// TwinCAT 3 PLC project plc_kfe_xgmd_vac
// ProgramVersion: 3.1.4022.3
// libraries:
//   L2SI Vacuum Library, * (SLAC)
//   LCLS General, * (SLAC)
//   Tc2_ControllerToolbox, * (Beckhoff Automation GmbH)
//   Tc2_MC2, * (Beckhoff Automation GmbH)
//   Tc2_Standard, * (Beckhoff Automation GmbH)
//   Tc2_System, * (Beckhoff Automation GmbH)
//   Tc2_Utilities, * (Beckhoff Automation GmbH)
//   Tc3_Module, * (Beckhoff Automation GmbH)
// project tree:
//   DUTs/ E_GasType.TcDUT, E_HomeState.TcDUT, E_MoveState.TcDUT (not stored), ST_HV.TcDUT (not stored), ST_VGP.TcDUT
//   GVLs/ GVL_Devices.TcGVL (not stored), GVL_GMD.TcGVL (not stored), GVL_VARIABLES.TcGVL (not stored)
//   / PlcTask.TcTTO (not stored)
//   POUs/ FB_HighVoltage.TcPOU, FB_VGP.TcPOU, MAIN.TcPOU (not stored), PRG_DIAGNOSTIC.TcPOU (not stored), PRG_Gas_Selection.TcPOU, PRG_GMD.TcPOU (not stored), PRG_HV_ILK.TcPOU (not stored), PRG_INJ.TcPOU, PRG_PressureControl.TcPOU (not stored), PRG_Purge.TcPOU, PRG_VGP.TcPOU
// real-time tasks:
//   TASK PlcTask: cycle T#10ms, priority 20, ADS port 350
//   TASK SimTask: cycle T#5ms, priority 21, ADS port 351
// motion (NC):
//   TASK NC-Task 1 SAF: cycle T#2ms, priority 4, ADS port 501
//   TASK NC-Task 1 SVB: cycle T#10ms, priority 8, ADS port 511
//   AXIS VGP_50 (id 1)
//     General: UnitName=step
//     Velo: Maximum=21000
//     OtherSettings: AllowMotionCmdToSlave=true
//     encoder EncType=4
//       EncPara: ScaleFactorNumerator=0.0390625, Inverse=true, MaxCount=#x0000ffff
//         SoftEndMinControl: Enable=true, Range=-15
//         SoftEndMaxControl: Enable=true, Range=1670
//         Inc: RefSoftSyncMask=#x0000ffff
//     drive DrvType=24
//       Analog: VeloReferenz=2000, ScaleFactorActTorque=0.1
//       TimeComp: TaskDelayCycles=1
//     controller CtrType=1
//       CtrPara: PriorControlFactor=1
//         PosDiffControl: Range=50
//         Observer: BandWidth=20
// I/O:
//   DEVICE Device 1 (EtherCAT), AmsNetId 5.62.5.76.2.1
//     EK1200_00_00 [EK1200-5000 EtherCAT Power supply (2A E-Bus)]
//       EL2202_00_01 [EL2202 2Ch. Dig. Output 24V, 0.5A]
//       EL3064_00_02 [EL3064 4Ch. Ana. Input 0-10V]
//       EL1008 [EL1008 8Ch. Dig. Input 24V, 3ms]
//       Term 28 (EL2008) [EL2008 8Ch. Dig. Output 24V, 0.5A]
//       Term 29 (EL2794) [EL2794 4Ch. Dig. Output 24V AC/DC, 2A, short-circuit-proof]
//       Term 30 (EL6695) [EL6695 EtherCAT Bridge terminal (Primary)]
//       Term 31 (EL6695) [EL6695 EtherCAT Bridge terminal (Primary)]
//       Term 32 (EK1110) [EK1110 EtherCAT extension]
//     EK1100_01_00 [EK1100 EtherCAT Coupler (2A E-Bus)]
//       EL3068_01_01 [EL3068 8Ch. Ana. Input 0-10V]
//       EL2794_01_02 [EL2794 4Ch. Dig. Output 24V AC/DC, 2A, short-circuit-proof]
//       EL2794_01_04 [EL2794 4Ch. Dig. Output 24V AC/DC, 2A, short-circuit-proof]
//       EL3068_01_05 [EL3068 8Ch. Ana. Input 0-10V]
//       EL3068_01_06 [EL3068 8Ch. Ana. Input 0-10V]
//       EL2794_01_07 [EL2794 4Ch. Dig. Output 24V AC/DC, 2A, short-circuit-proof]
//       EL2794_01_09 [EL2794 4Ch. Dig. Output 24V AC/DC, 2A, short-circuit-proof]
//       EL3068_01_10 [EL3068 8Ch. Ana. Input 0-10V]
//       EL3068_01_11 [EL3068 8Ch. Ana. Input 0-10V]
//       EL2794_01_12 [EL2794 4Ch. Dig. Output 24V AC/DC, 2A, short-circuit-proof]
//       EL2794_01_14 [EL2794 4Ch. Dig. Output 24V AC/DC, 2A, short-circuit-proof]
//       EL3068_01_15 [EL3068 8Ch. Ana. Input 0-10V]
//       EK1110_01_16 [EK1110 EtherCAT extension]
//     EK1100_02_00 [EK1100 EtherCAT Coupler (2A E-Bus)]
//       EL2004_02_01 [EL2004 4Ch. Dig. Output 24V, 0.5A]
//       EL1004_02_02 [EL1004 4Ch. Dig. Input 24V, 3ms]
//       EL2004_02_03 [EL2004 4Ch. Dig. Output 24V, 0.5A]
//       EL1088_02_04 [EL1088 8Ch. Dig. Input 24V, 3ms, negative]
//       EL2004_02_05 [EL2004 4Ch. Dig. Output 24V, 0.5A]
//       EL1088_02_06 [EL1088 8Ch. Dig. Input 24V, 3ms, negative]
//       EL2004_02_07 [EL2004 4Ch. Dig. Output 24V, 0.5A]
//       EL1004_02_08 [EL1004 4Ch. Dig. Input 24V, 3ms]
//       EL2004_02_09 [EL2004 4Ch. Dig. Output 24V, 0.5A]
//       EL1088_02_10 [EL1088 8Ch. Dig. Input 24V, 3ms, negative]
//       EL2004_02_11 [EL2004 4Ch. Dig. Output 24V, 0.5A]
//       EL1004_02_13 [EL1004 4Ch. Dig. Input 24V, 3ms]
//       EL2004_02_14 [EL2004 4Ch. Dig. Output 24V, 0.5A]
//       EL1088_02_15 [EL1088 8Ch. Dig. Input 24V, 3ms, negative]
//       EL2004_02_16 [EL2004 4Ch. Dig. Output 24V, 0.5A]
//       EL1004_02_17 [EL1004 4Ch. Dig. Input 24V, 3ms]
//       EL3064_02_18 [EL3064 4Ch. Ana. Input 0-10V]
//       EL1008_02_20 [EL1008 8Ch. Dig. Input 24V, 3ms]
//       EL2008_02_22 [EL2008 8Ch. Dig. Output 24V, 0.5A]
//       EL2794_02_23 [EL2794 4Ch. Dig. Output 24V AC/DC, 2A, short-circuit-proof]
//       EL1004_02_24 [EL1004 4Ch. Dig. Input 24V, 3ms]
//       EL2794_02_25 [EL2794 4Ch. Dig. Output 24V AC/DC, 2A, short-circuit-proof]
//       Term 70 (EL9011) [EL9011 End Terminal]
//     EK1100_03_00 (EK1100) [EK1100 EtherCAT Coupler (2A E-Bus)]
//       EL4004_03_01 [EL4004 4Ch. Ana. Output 0-10V, 12bit]
//       EL7041_03_02 [EL7041 1Ch. Stepper motor output stage (50V, 5A)]
//       EL5101_03_03 [EL5101 1Ch. Inc. Encoder 5V]
//       EL1004_03_04 [EL1004 4Ch. Dig. Input 24V, 3ms]
//       EL2004_03_05 [EL2004 4Ch. Dig. Output 24V, 0.5A]
//       EL2004_03_06 [EL2004 4Ch. Dig. Output 24V, 0.5A]
//       EL2004_03_07 [EL2004 4Ch. Dig. Output 24V, 0.5A]
//       EL3202_03_08 [EL3202 2Ch. Ana. Input PT100 (RTD)]
//       EL3174_03_09 [EL3174-0002 4Ch. Ana. Input +/-10V, +/-20mA 16 Bit, Isolated Channels]
// variable links:
//   NC-Task 1 SAF/Axes/VGP_50 <-> Device 1 (EtherCAT)/EK1100_03_00 (EK1100)/EL5101_03_03
//     Enc/Inputs/In/nDataIn1[0] <-> ENC Status compact/Counter value
//     Enc/Inputs/In/nDataIn2[0] <-> ENC Status compact/Latch value
//     Enc/Inputs/In/nState1 @bit 4 <-> ENC Status compact/Status/Counter overflow
//     Enc/Inputs/In/nState1 @bit 3 <-> ENC Status compact/Status/Counter underflow
//     Enc/Inputs/In/nState1 @bit 7 <-> ENC Status compact/Status/Extrapolation stall
//     Enc/Inputs/In/nState1 <-> ENC Status compact/Status/Latch C valid
//     Enc/Inputs/In/nState1 @bit 1 <-> ENC Status compact/Status/Latch extern valid
//     Enc/Inputs/In/nState1 @bit 6 <-> ENC Status compact/Status/Open circuit
//     Enc/Inputs/In/nState1 @bit 2 <-> ENC Status compact/Status/Set counter done
//     Enc/Inputs/In/nState1 @bit 5 <-> ENC Status compact/Status/Status of input status
//     Enc/Inputs/In/nState2 @bit 4 <-> ENC Status compact/Status/Status of extern latch
//     Enc/Inputs/In/nState2 <-> ENC Status compact/Status/Status of input A
//     Enc/Inputs/In/nState2 @bit 1 <-> ENC Status compact/Status/Status of input B
//     Enc/Inputs/In/nState2 @bit 2 <-> ENC Status compact/Status/Status of input C
//     Enc/Inputs/In/nState2 @bit 3 <-> ENC Status compact/Status/Status of input gate
//     Enc/Inputs/In/nState2 @bit 5 <-> ENC Status compact/Status/Sync error
//     Enc/Inputs/In/nState2 @bit 6 <-> ENC Status compact/Status/TxPDO State
//     Enc/Inputs/In/nState2 @bit 7 <-> ENC Status compact/Status/TxPDO Toggle
//     Enc/Inputs/In/nState4 @bit 1 <-> WcState/InputToggle
//     Enc/Inputs/In/nState4 <-> WcState/WcState
//     Enc/Outputs/Out/nCtrl1 <-> ENC Control compact/Control/Enable latch C
//     Enc/Outputs/Out/nCtrl1 @bit 3 <-> ENC Control compact/Control/Enable latch extern on negative edge
//     Enc/Outputs/Out/nCtrl1 @bit 1 <-> ENC Control compact/Control/Enable latch extern on positive edge
//     Enc/Outputs/Out/nCtrl1 @bit 2 <-> ENC Control compact/Control/Set counter
//     Enc/Outputs/Out/nDataOut1[0] <-> ENC Control compact/Set counter value
//   NC-Task 1 SAF/Axes/VGP_50 <-> Device 1 (EtherCAT)/EK1100_03_00 (EK1100)/EL7041_03_02
//     Drive/Inputs/In/nState1 @bit 3 <-> STM Status/Status/Error
//     Drive/Inputs/In/nState1 @bit 5 <-> STM Status/Status/Moving negative
//     Drive/Inputs/In/nState1 @bit 4 <-> STM Status/Status/Moving positive
//     Drive/Inputs/In/nState1 @bit 1 <-> STM Status/Status/Ready
//     Drive/Inputs/In/nState1 <-> STM Status/Status/Ready to enable
//     Drive/Inputs/In/nState1 @bit 6 <-> STM Status/Status/Torque reduced
//     Drive/Inputs/In/nState1 @bit 2 <-> STM Status/Status/Warning
//     Drive/Inputs/In/nState2 @bit 3 <-> STM Status/Status/Digital input 1
//     Drive/Inputs/In/nState2 @bit 4 <-> STM Status/Status/Digital input 2
//     Drive/Inputs/In/nState2 @bit 5 <-> STM Status/Status/Sync error
//     Drive/Inputs/In/nState2 @bit 7 <-> STM Status/Status/TxPDO Toggle
//     Drive/Inputs/In/nState4 @bit 1 <-> WcState/InputToggle
//     Drive/Inputs/In/nState4 <-> WcState/WcState
//     Drive/Outputs/Out/nCtrl1 <-> STM Control/Control/Enable
//     Drive/Outputs/Out/nCtrl1 @bit 2 <-> STM Control/Control/Reduce torque
//     Drive/Outputs/Out/nCtrl1 @bit 1 <-> STM Control/Control/Reset
//     Drive/Outputs/Out/nDataOut2[0] <-> STM Velocity/Velocity
//   plc_kfe_xgmd_vac/plc_kfe_xgmd_vac Instance <-> Device 1 (EtherCAT)/EK1100_01_00/EL2794_01_02
//     PlcTask Outputs/GVL_GMD.fb_EM2K0_XGMD_GCC_10.q_xHV_DIS <-> Channel 1/Output
//     PlcTask Outputs/GVL_GMD.fb_EM2K0_XGMD_GCC_20.q_xHV_DIS <-> Channel 2/Output
//     PlcTask Outputs/GVL_GMD.fb_EM2K0_XGMD_GCC_30.q_xHV_DIS <-> Channel 3/Output
//   plc_kfe_xgmd_vac/plc_kfe_xgmd_vac Instance <-> Device 1 (EtherCAT)/EK1100_01_00/EL2794_01_04
//     PlcTask Outputs/GVL_GMD.fb_EM2K0_XGMD_GCC_40.q_xHV_DIS <-> Channel 1/Output
//     PlcTask Outputs/GVL_GMD.fb_EM2K0_XGMD_GCC_50.q_xHV_DIS <-> Channel 2/Output
//   plc_kfe_xgmd_vac/plc_kfe_xgmd_vac Instance <-> Device 1 (EtherCAT)/EK1100_01_00/EL2794_01_07
//     PlcTask Outputs/GVL_GMD.fb_EM2K0_XGMD_GCC_60.q_xHV_DIS <-> Channel 1/Output
//     PlcTask Outputs/GVL_GMD.fb_EM2K0_XGMD_GCC_70.q_xHV_DIS <-> Channel 2/Output
//     PlcTask Outputs/GVL_GMD.fb_EM2K0_XGMD_GCC_80.q_xHV_DIS <-> Channel 3/Output
//   plc_kfe_xgmd_vac/plc_kfe_xgmd_vac Instance <-> Device 1 (EtherCAT)/EK1100_01_00/EL2794_01_09
//     PlcTask Outputs/GVL_GMD.fb_EM2K0_XGMD_GCC_90.q_xHV_DIS <-> Channel 1/Output
//   plc_kfe_xgmd_vac/plc_kfe_xgmd_vac Instance <-> Device 1 (EtherCAT)/EK1100_01_00/EL3068_01_01
//     PlcTask Inputs/GVL_GMD.fb_EM2K0_XGMD_GCC_10.i_iPRESS_R <-> AI Standard Channel 1/Value
//     PlcTask Inputs/GVL_GMD.fb_EM2K0_XGMD_GCC_20.i_iPRESS_R <-> AI Standard Channel 3/Value
//     PlcTask Inputs/GVL_GMD.fb_EM2K0_XGMD_GCC_30.i_iPRESS_R <-> AI Standard Channel 5/Value
//   plc_kfe_xgmd_vac/plc_kfe_xgmd_vac Instance <-> Device 1 (EtherCAT)/EK1100_01_00/EL3068_01_05
//     PlcTask Inputs/GVL_GMD.fb_EM2K0_XGMD_GCC_40.i_iPRESS_R <-> AI Standard Channel 1/Value
//     PlcTask Inputs/GVL_GMD.fb_EM2K0_XGMD_GCC_50.i_iPRESS_R <-> AI Standard Channel 3/Value
//     PlcTask Inputs/GVL_GMD.fb_EM2K0_XGMD_GPI_10.i_iPRESS_R <-> AI Standard Channel 5/Value
//     PlcTask Inputs/GVL_GMD.fb_EM2K0_XGMD_GPI_90.i_iPRESS_R <-> AI Standard Channel 6/Value
//   plc_kfe_xgmd_vac/plc_kfe_xgmd_vac Instance <-> Device 1 (EtherCAT)/EK1100_01_00/EL3068_01_06
//     PlcTask Inputs/GVL_GMD.fb_EM2K0_XGMD_GCC_60.i_iPRESS_R <-> AI Standard Channel 1/Value
//     PlcTask Inputs/GVL_GMD.fb_EM2K0_XGMD_GCC_70.i_iPRESS_R <-> AI Standard Channel 3/Value
//     PlcTask Inputs/GVL_GMD.fb_EM2K0_XGMD_GCC_80.i_iPRESS_R <-> AI Standard Channel 5/Value
//   plc_kfe_xgmd_vac/plc_kfe_xgmd_vac Instance <-> Device 1 (EtherCAT)/EK1100_01_00/EL3068_01_10
//     PlcTask Inputs/GVL_GMD.fb_EM2K0_XGMD_GCC_90.i_iPRESS_R <-> AI Standard Channel 1/Value
//     PlcTask Inputs/GVL_GMD.fb_EM2K0_XGMD_GPI_50.i_iPRESS_R <-> AI Standard Channel 5/Value
//   plc_kfe_xgmd_vac/plc_kfe_xgmd_vac Instance <-> Device 1 (EtherCAT)/EK1100_02_00/EL1004_02_02
//     PlcTask Inputs/GVL_GMD.fb_EM2K0_XGMD_VRC_10.i_xClsLS <-> Channel 2/Input
//     PlcTask Inputs/GVL_GMD.fb_EM2K0_XGMD_VRC_20.i_xClsLS <-> Channel 4/Input
//     PlcTask Inputs/GVL_GMD.fb_EM2K0_XGMD_VRC_10.i_xOpnLS <-> Channel 1/Input
//     PlcTask Inputs/GVL_GMD.fb_EM2K0_XGMD_VRC_20.i_xOpnLS <-> Channel 3/Input
//   plc_kfe_xgmd_vac/plc_kfe_xgmd_vac Instance <-> Device 1 (EtherCAT)/EK1100_02_00/EL1004_02_08
//     PlcTask Inputs/GVL_GMD.fb_EM2K0_XGMD_VRC_30.i_xClsLS <-> Channel 2/Input
//     PlcTask Inputs/GVL_GMD.fb_EM2K0_XGMD_VRC_40.i_xClsLS <-> Channel 4/Input
//     PlcTask Inputs/GVL_GMD.fb_EM2K0_XGMD_VRC_30.i_xOpnLS <-> Channel 1/Input
//     PlcTask Inputs/GVL_GMD.fb_EM2K0_XGMD_VRC_40.i_xOpnLS <-> Channel 3/Input
//   plc_kfe_xgmd_vac/plc_kfe_xgmd_vac Instance <-> Device 1 (EtherCAT)/EK1100_02_00/EL1004_02_13
//     PlcTask Inputs/GVL_GMD.fb_EM2K0_XGMD_VRC_60.i_xClsLS <-> Channel 2/Input
//     PlcTask Inputs/GVL_GMD.fb_EM2K0_XGMD_VRC_70.i_xClsLS <-> Channel 4/Input
//     PlcTask Inputs/GVL_GMD.fb_EM2K0_XGMD_VRC_60.i_xOpnLS <-> Channel 1/Input
//     PlcTask Inputs/GVL_GMD.fb_EM2K0_XGMD_VRC_70.i_xOpnLS <-> Channel 3/Input
//   plc_kfe_xgmd_vac/plc_kfe_xgmd_vac Instance <-> Device 1 (EtherCAT)/EK1100_02_00/EL1004_02_17
//     PlcTask Inputs/GVL_GMD.fb_EM2K0_XGMD_VRC_80.i_xClsLS <-> Channel 2/Input
//     PlcTask Inputs/GVL_GMD.fb_EM2K0_XGMD_VRC_90.i_xClsLS <-> Channel 4/Input
//     PlcTask Inputs/GVL_GMD.fb_EM2K0_XGMD_VRC_80.i_xOpnLS <-> Channel 1/Input
//     PlcTask Inputs/GVL_GMD.fb_EM2K0_XGMD_VRC_90.i_xOpnLS <-> Channel 3/Input
//   plc_kfe_xgmd_vac/plc_kfe_xgmd_vac Instance <-> Device 1 (EtherCAT)/EK1100_02_00/EL1004_02_24
//     PlcTask Inputs/GVL_GMD.fb_EM2K0_XGMD_PRT_50.i_xAlarmOK <-> Channel 2/Input
//     PlcTask Inputs/GVL_GMD.fb_EM2K0_XGMD_PRT_50.i_xIsRun <-> Channel 1/Input
//   plc_kfe_xgmd_vac/plc_kfe_xgmd_vac Instance <-> Device 1 (EtherCAT)/EK1100_02_00/EL1088_02_04
//     PlcTask Inputs/GVL_GMD.fb_EM2K0_XGMD_PTM_10.i_xAtSpd <-> Channel 1/Input
//     PlcTask Inputs/GVL_GMD.fb_EM2K0_XGMD_PTM_20.i_xAtSpd <-> Channel 3/Input
//     PlcTask Inputs/GVL_GMD.fb_EM2K0_XGMD_PTM_10.i_xFault <-> Channel 2/Input
//     PlcTask Inputs/GVL_GMD.fb_EM2K0_XGMD_PTM_20.i_xFault <-> Channel 4/Input
//   plc_kfe_xgmd_vac/plc_kfe_xgmd_vac Instance <-> Device 1 (EtherCAT)/EK1100_02_00/EL1088_02_06
//     PlcTask Inputs/GVL_GMD.fb_EM2K0_XGMD_PTM_30.i_xAtSpd <-> Channel 1/Input
//     PlcTask Inputs/GVL_GMD.fb_EM2K0_XGMD_PTM_40.i_xAtSpd <-> Channel 3/Input
//     PlcTask Inputs/GVL_GMD.fb_EM2K0_XGMD_PTM_50.i_xAtSpd <-> Channel 5/Input
//     PlcTask Inputs/GVL_GMD.fb_EM2K0_XGMD_PTM_30.i_xFault <-> Channel 2/Input
//     PlcTask Inputs/GVL_GMD.fb_EM2K0_XGMD_PTM_40.i_xFault <-> Channel 4/Input
//     PlcTask Inputs/GVL_GMD.fb_EM2K0_XGMD_PTM_50.i_xFault <-> Channel 6/Input
//   plc_kfe_xgmd_vac/plc_kfe_xgmd_vac Instance <-> Device 1 (EtherCAT)/EK1100_02_00/EL1088_02_10
//     PlcTask Inputs/GVL_GMD.fb_EM2K0_XGMD_PTM_60.i_xAtSpd <-> Channel 1/Input
//     PlcTask Inputs/GVL_GMD.fb_EM2K0_XGMD_PTM_70.i_xAtSpd <-> Channel 3/Input
//     PlcTask Inputs/GVL_GMD.fb_EM2K0_XGMD_PTM_60.i_xFault <-> Channel 2/Input
//     PlcTask Inputs/GVL_GMD.fb_EM2K0_XGMD_PTM_70.i_xFault <-> Channel 4/Input
//   plc_kfe_xgmd_vac/plc_kfe_xgmd_vac Instance <-> Device 1 (EtherCAT)/EK1100_02_00/EL1088_02_15
//     PlcTask Inputs/GVL_GMD.fb_EM2K0_XGMD_PTM_80.i_xAtSpd <-> Channel 1/Input
//     PlcTask Inputs/GVL_GMD.fb_EM2K0_XGMD_PTM_90.i_xAtSpd <-> Channel 3/Input
//     PlcTask Inputs/GVL_GMD.fb_EM2K0_XGMD_PTM_80.i_xFault <-> Channel 2/Input
//     PlcTask Inputs/GVL_GMD.fb_EM2K0_XGMD_PTM_90.i_xFault <-> Channel 4/Input
//   plc_kfe_xgmd_vac/plc_kfe_xgmd_vac Instance <-> Device 1 (EtherCAT)/EK1100_02_00/EL2004_02_01
//     PlcTask Outputs/GVL_GMD.fb_EM2K0_XGMD_VRC_10.q_xOPN_DO <-> Channel 1/Output
//     PlcTask Outputs/GVL_GMD.fb_EM2K0_XGMD_VRC_20.q_xOPN_DO <-> Channel 3/Output
//   plc_kfe_xgmd_vac/plc_kfe_xgmd_vac Instance <-> Device 1 (EtherCAT)/EK1100_02_00/EL2004_02_03
//     PlcTask Outputs/GVL_GMD.fb_EM2K0_XGMD_PTM_10.q_RunDO <-> Channel 1/Output
//     PlcTask Outputs/GVL_GMD.fb_EM2K0_XGMD_PTM_20.q_RunDO <-> Channel 2/Output
//   plc_kfe_xgmd_vac/plc_kfe_xgmd_vac Instance <-> Device 1 (EtherCAT)/EK1100_02_00/EL2004_02_05
//     PlcTask Outputs/GVL_GMD.fb_EM2K0_XGMD_PTM_30.q_RunDO <-> Channel 1/Output
//     PlcTask Outputs/GVL_GMD.fb_EM2K0_XGMD_PTM_40.q_RunDO <-> Channel 2/Output
//     PlcTask Outputs/GVL_GMD.fb_EM2K0_XGMD_PTM_50.q_RunDO <-> Channel 3/Output
//   plc_kfe_xgmd_vac/plc_kfe_xgmd_vac Instance <-> Device 1 (EtherCAT)/EK1100_02_00/EL2004_02_07
//     PlcTask Outputs/GVL_GMD.fb_EM2K0_XGMD_VRC_30.q_xOPN_DO <-> Channel 1/Output
//     PlcTask Outputs/GVL_GMD.fb_EM2K0_XGMD_VRC_40.q_xOPN_DO <-> Channel 3/Output
//   plc_kfe_xgmd_vac/plc_kfe_xgmd_vac Instance <-> Device 1 (EtherCAT)/EK1100_02_00/EL2004_02_09
//     PlcTask Outputs/GVL_GMD.fb_EM2K0_XGMD_PTM_60.q_RunDO <-> Channel 1/Output
//     PlcTask Outputs/GVL_GMD.fb_EM2K0_XGMD_PTM_70.q_RunDO <-> Channel 2/Output
//   plc_kfe_xgmd_vac/plc_kfe_xgmd_vac Instance <-> Device 1 (EtherCAT)/EK1100_02_00/EL2004_02_11
//     PlcTask Outputs/GVL_GMD.fb_EM2K0_XGMD_VRC_60.q_xOPN_DO <-> Channel 1/Output
//     PlcTask Outputs/GVL_GMD.fb_EM2K0_XGMD_VRC_70.q_xOPN_DO <-> Channel 3/Output
//   plc_kfe_xgmd_vac/plc_kfe_xgmd_vac Instance <-> Device 1 (EtherCAT)/EK1100_02_00/EL2004_02_14
//     PlcTask Outputs/GVL_GMD.fb_EM2K0_XGMD_PTM_80.q_RunDO <-> Channel 1/Output
//     PlcTask Outputs/GVL_GMD.fb_EM2K0_XGMD_PTM_90.q_RunDO <-> Channel 2/Output
//   plc_kfe_xgmd_vac/plc_kfe_xgmd_vac Instance <-> Device 1 (EtherCAT)/EK1100_02_00/EL2004_02_16
//     PlcTask Outputs/GVL_GMD.fb_EM2K0_XGMD_VRC_80.q_xOPN_DO <-> Channel 1/Output
//     PlcTask Outputs/GVL_GMD.fb_EM2K0_XGMD_VRC_90.q_xOPN_DO <-> Channel 3/Output
//   plc_kfe_xgmd_vac/plc_kfe_xgmd_vac Instance <-> Device 1 (EtherCAT)/EK1100_02_00/EL2794_02_25
//     PlcTask Outputs/GVL_GMD.fb_EM2K0_XGMD_PRT_50.q_xRemote <-> Channel 2/Output
//     PlcTask Outputs/GVL_GMD.fb_EM2K0_XGMD_PRT_50.q_xRunDo <-> Channel 1/Output
//   plc_kfe_xgmd_vac/plc_kfe_xgmd_vac Instance <-> Device 1 (EtherCAT)/EK1100_03_00 (EK1100)/EL2004_03_06
//     PlcTask Outputs/GVL_Devices.VVC_{80..83}.q_xOPN_DO <-> Channel {1..4}/Output  (4 links)
//   plc_kfe_xgmd_vac/plc_kfe_xgmd_vac Instance <-> Device 1 (EtherCAT)/EK1100_03_00 (EK1100)/EL2004_03_07
//     PlcTask Outputs/GVL_Devices.VVC_84.q_xOPN_DO <-> Channel 1/Output
//     PlcTask Outputs/GVL_Devices.VVC_85.q_xOPN_DO <-> Channel 2/Output
//     PlcTask Outputs/GVL_Devices.VVC_86.q_xOPN_DO <-> Channel 3/Output
//   plc_kfe_xgmd_vac/plc_kfe_xgmd_vac Instance <-> Device 1 (EtherCAT)/EK1100_03_00 (EK1100)/EL3174_03_09
//     PlcTask Inputs/GVL_Devices.GCM_80.i_iPRESS_R <-> AI Standard Channel 1/Value
//     PlcTask Inputs/GVL_Devices.GHC_50.i_iPRESS_R <-> AI Standard Channel 2/Value
//   plc_kfe_xgmd_vac/plc_kfe_xgmd_vac Instance <-> Device 1 (EtherCAT)/EK1100_03_00 (EK1100)/EL4004_03_01
//     PlcTask Outputs/GVL_Devices.VCN_50.q_iRawPosition <-> AO Outputs Channel 1/Analog output

// ---- DUTs/E_GasType.TcDUT
TYPE E_GasType :
(
	none := 0,
	Neon,
	Argon,
	Krypton,
	Xenon
);
END_TYPE

// ---- DUTs/E_HomeState.TcDUT
TYPE E_HomeState :
(
	READY,
	INIT,
	MOVING,
	MOVING2,
	CHECK,
	ERROR,
	WRITE,
	DONE
	
) UDINT;
END_TYPE

// ---- DUTs/ST_VGP.TcDUT
TYPE ST_VGP :
STRUCT

	{attribute 'pytmc' := '
    pv: POS_RDBK;
	io: i;
    '}
	// Inputs
	i_iPosition	:	REAL; //Encoder position readback (if it exists)
	{attribute 'pytmc' := '
    pv: ENC_RDBK;
	io: i;
    '}
	// Inputs
	rEnoder_Position	:	REAL; //Encoder position readback (if it exists)
	{attribute 'pytmc' := '
    pv: ERROR;
	io: i;
    '}
	// Inputs
	pv_xError	:	BOOL;
	
	{attribute 'pytmc' := '
    pv: IS_HOMED;
	io: i;
    '}
	// Inputs
	pv_xHomed	:	BOOL :=false;
	
	//Softvariables
	{attribute 'pytmc' := '
    pv: ILK_OK;
	io: i;
    '}
	xIlkOK	:	BOOL := FALSE; // Interlock Bit
	//Manually Pressing valve "Open/Close" on EDM
	{attribute 'pytmc' := '
    pv: OPN_SW;
	io: io;
    '}
	pv_xOPN_SW	: BOOL;
	
	{attribute 'pytmc' := '
    pv: GO_SW;
	io: io;
    '}
	pv_xGo_SW	: BOOL;
	
	{attribute 'pytmc' := '
    pv: HOME_SW;
	io: io;
    '}
	pv_xHome_SW	: BOOL;
	
	{attribute 'pytmc' := '
    pv: ABORT;
	io: io;
    '}
	pv_xABORT_SW	: BOOL;
	
	rUpperLimit	:	REAL:=100;	//Percentage Upper limit on valve open
	{attribute 'pytmc' := '
	pv: POS_CTRL;
	io: io; 
	'}
	rReqPosition	:	REAL; 
	// Outputs
	{attribute 'pytmc' := '
	pv: POS_DES;
	io: io;
	'}
	q_iRawPosition	:	INT; //Position control 
	{attribute 'pytmc' := '
	pv: STATE;
	io: io;
	'}
	eValveControl	:	E_VCN := CloseValve; // Valve control state
	/// state machine state 
	{attribute 'pytmc' := '
	pv: STATE;
	io: io;
	'}
	state: E_MoveState; //Axis Move state
	ftIlk	:	F_TRIG;	

END_STRUCT
END_TYPE

// ---- POUs/FB_HighVoltage.TcPOU
FUNCTION_BLOCK FB_HighVoltage
VAR_INPUT
	i_xExtIlkOK	:	BOOL; //External Interlock, SET to TRUE if not used
END_VAR
VAR_OUTPUT
	{attribute 'pytmc' := '
    pv:
	'}
	hv:ST_HV;
END_VAR
VAR
	(*outputs*)
	q_HV_DO AT %Q*: BOOL;
END_VAR


hv.xIlkOK := i_xExtIlkOK;

q_HV_DO := hv.HV_sw AND hv.xIlkOK;

(*soft io mapping*)
hv.q_HV_DO := q_HV_DO;

END_FUNCTION_BLOCK

// ---- POUs/FB_VGP.TcPOU
(* This function implements the Basic functions for the Vat Motorized valve*)
FUNCTION_BLOCK FB_VGP
VAR_INPUT
	i_xExtIlkOK	:	BOOL; //External Interlock, SET to TRUE if not used
	i_ReqPos	:	REAL; //Requested position
	
	arrTable	: ARRAY[1..14,1..2] OF FLOAT;
END_VAR
VAR_OUTPUT
	{attribute 'pytmc' := '
    pv:
	'}
	q_stVGP	:	ST_VGP; // valve structure
END_VAR
VAR_IN_OUT
	
END_VAR

VAR CONSTANT
	
	rClosePosition : REAL:=0; // Encoder Min. Fully Closed
	rMaxDiffPressure: REAL:= 22.5; //Torr
END_VAR

VAR
	rOpenPosition: REAL:=1645; // Encoder MAX. Fully Open
	rTargetPosition : REAL;
	rTargetVelocity: REAL:=30;
	rHomingVelocity: REAL:=10;
	rHomingDistance: REAL:=20;//every 150 is 10% , 1%  is 14.975
	rOldTargetPosition: REAL;
		
	// 
	/// axis reference data structure 
	Axis: AXIS_REF;
	//
	InfoData_State AT %I*: UINT ;
	
	// Axis MC functions

	fbPowerAxis: MC_Power;
	/// debug function block output data 
	PowerAxisOut: ST_McOutputs;
	fbMoveAxisABS: MC_MoveAbsolute;
	/// debug function block output data 
	MoveAbsoluteOut: ST_McOutputs;
	fbMoveAxisABS2: MC_MoveAbsolute;
	/// debug function block output data 
	MoveAbsoluteOut2: ST_McOutputs;
	
	fbReset: MC_Reset;
	/// debug function block output data 
	ResetOut: ST_McOutputs;
	MoveAxisREL: MC_MoveAbsolute;
	MoveRelativeOut: ST_McOutputs;
	
	
	nErrorID: UDINT;
	bError : Bool;
	sErrorMessage : STRING;
	rOverride: LREAL := 100;
	fbHalt: MC_Halt;
	
	
	// Homing Functions
	bGo:BOOL := FALSE; //to execute motion
	bHome:BOOL :=FALSE; // should be set to true
	bEnable:Bool; //to be removed
	fbMoveRel: MC_MoveRelative;
	fbSetPosition: MC_SetPosition;
	fbWriteParameter: MC_WriteBoolParameter;
	HomeState: E_HomeState;
	
	
	// interpolation
	bInit : BOOL := TRUE;
	eMode           : E_CTRL_MODE;
	iCounter:INT;
	//CONTROL
	stCTRL_LIN_INTERPOLATION_PARAMS		: ST_CTRL_LIN_INTERPOLATION_PARAMS;
	fbCTRL_LIN_INTERPOLATION					: FB_CTRL_LIN_INTERPOLATION;
	arrTable_ENC : ARRAY[1..14,1..2] OF FLOAT;
	//Readdback
	stCTRL_LIN_INTERPOLATION_PARAMS_ENC		: ST_CTRL_LIN_INTERPOLATION_PARAMS;
	fbCTRL_LIN_INTERPOLATION_ENC					: FB_CTRL_LIN_INTERPOLATION;

END_VAR

/// Interpolation  function initialization
ACT_INIT();

// Interlocking
q_stVGP.xIlkOK := i_xExtIlkOK;
(*Checking which Control mode is selected*)
IF q_stVGP.xIlkOK AND NOT (q_stVGP.pv_xError) THEN
	IF q_stVGP.eValveControl = OpenValve THEN
		q_stVGP.rReqPosition := q_stVGP.rUpperLimit;
	ELSIF q_stVGP.eValveControl = CloseValve THEN
		q_stVGP.rReqPosition := 0;
	ELSIF q_stVGP.eValveControl = ManualControl THEN
		q_stVGP.rReqPosition := LIMIT(0, q_stVGP.rReqPosition, q_stVGP.rUpperLimit);
	ELSIF q_stVGP.eValveControl = PressureControl THEN
		 q_stVGP.rReqPosition := LIMIT(0, i_ReqPos, q_stVGP.rUpperLimit);
	END_IF
ELSE
	q_stVGP.rReqPosition := 0;
	q_stVGP.eValveControl := CloseValve;//CloseValve;
	bGo:=FALSE;
END_IF


//Check the Drive State

IF (*(InfoData_State<>16#8) OR*) (q_stVGP.state = MOVESTATE_ERROR) THEN
	q_stVGP.pv_xError:=TRUE;
ELSE
	q_stVGP.pv_xError:=FALSE;
	// Call function to execute move
	// call motion function blocks???
END_IF


IF (q_stVGP.pv_xABORT_SW ) THEN
	q_stVGP.pv_xABORT_SW := FALSE;
	q_stVGP.state:= MOVESTATE_ABORT;
END_IF


ACT_LIN_INTERPOLATION();
ACT_AXIS();
//ACT_HOME();

ACTION ACT_AXIS:
//update the axis status
AXIS();
q_stVGP.rEnoder_Position := LREAL_TO_REAL(Axis.NcToPlc.ActPos); // encoder position

//Homing STATE is missing

// state machine for axis motion
	(* move axis using a state machine *)
	CASE q_stVGP.state OF

		MOVESTATE_INIT :	(* initialisation *)
			(* initialize all function blocks *)
			fbMoveAxisABS.Execute := FALSE;
			fbMoveAxisABS2.Execute := FALSE;
			fbReset.Execute := FALSE;
			fbHALT.Execute :=FALSE;//
			q_stVGP.state := MOVESTATE_ENABLE; // Check homing first

		MOVESTATE_ENABLE :
			fbPowerAxis.Enable :=  TRUE;
			fbPowerAxis.Enable_Positive := TRUE;
			fbPowerAxis.Enable_Negative := TRUE;
			IF fbPowerAxis.Status THEN
				q_stVGP.state := MOVESTATE_READY;
			ELSIF fbPowerAxis.Error THEN
				q_stVGP.state := MOVESTATE_ERROR;
			END_IF
		
		MOVESTATE_READY: // waiting for move command
			IF (HomeState = READY) AND (q_stVGP.pv_xHome_SW) THEN
					HomeState:= INIT;
					q_stVGP.pv_xHome_SW:=false;
					bHome := false;
					q_stVGP.state := MOVESTATE_HOME;
					ELSE 
					q_stVGP.state := MOVESTATE_READY;
				END_IF
			IF (q_stVGP.pv_xGo_SW) AND i_xExtIlkOK(* AND( rOldTargetPosition <> rTargetPosition) *) THEN
				q_stVGP.pv_xGo_SW := false;
				q_stVGP.state := MOVESTATE_NEWTARGETPOSITION;	
			END_IF
			IF NOT fbPowerAxis.Status THEN
				q_stVGP.state := MOVESTATE_ENABLE;
			ELSIF fbPowerAxis.Error THEN
				q_stVGP.state := MOVESTATE_ERROR;
			END_IF
			
		MOVESTATE_HOME:
				if (HomeState = DONE) THEN
					 q_stVGP.state := MOVESTATE_READY;
					 q_stVGP.pv_xHomed := TRUE;
				END_IF
				
				if (HomeState = ERROR) THEN
					 q_stVGP.state := MOVESTATE_ERROR;
					  q_stVGP.pv_xHomed := FALSE;
				END_IF
				
		MOVESTATE_NEWTARGETPOSITION:
			fbMoveAxisABS.Position := rTargetPosition;	
			fbMoveAxisABS.Velocity := rTargetVelocity;		
			//fbMoveAxisABS.BufferMode := MC_BlendingNext;
			fbMoveAxisABS.Execute := TRUE;
			IF fbMoveAxisABS.Active  THEN
				(* axis is executing job but is not yet finished *)
				fbMoveAxisABS.Execute := FALSE;
				(* leave this state and buffer a second command *)
				q_stVGP.state := MOVESTATE_MOVING; 
			ElSIF fbMoveAxisABS.Done THEN
				fbMoveAxisABS.Execute := FALSE;
				q_stVGP.state := MOVESTATE_READY;
			ELSIF fbMoveAxisABS.CommandAborted OR fbMoveAxisABS.Error THEN
				q_stVGP.state := MOVESTATE_ERROR;
			END_IF
			
				
		MOVESTATE_MOVING://
			IF fbMoveAxisABS.CommandAborted OR fbMoveAxisABS.Error THEN
				q_stVGP.state := MOVESTATE_ERROR;
			END_IF	
			IF NOT ( Axis.Status.Moving) OR (fbMoveAxisABS.Done) THEN //(fbMoveAxisABS.Done) AND (fbMoveAxisABS2.Done) THEN
				q_stVGP.state := MOVESTATE_READY;	
			END_IF
			
		
		MOVESTATE_HALT:
			fbHALT.Execute :=TRUE;
			IF Axis.Status.Error THEN
				q_stVGP.state := MOVESTATE_RESET;	(* axis error requires reset *)
			ELSE
				q_stVGP.state := MOVESTATE_INIT;		(* function block errors don't need a reset *)
			END_IF
		
		MOVESTATE_ERROR :
			
			IF Axis.Status.Error THEN
				q_stVGP.state := MOVESTATE_RESET;	(* axis error requires reset *)
			ELSE
				q_stVGP.state := MOVESTATE_INIT;		(* function block errors don't need a reset *)
			END_IF

		MOVESTATE_RESET :
			fbReset.Execute := TRUE;
			IF fbReset.Done THEN
				q_stVGP.state := MOVESTATE_INIT;
			ELSIF fbReset.Error THEN
				q_stVGP.state := MOVESTATE_ERROR; (* keep trying to reset*)
			END_IF
			
		MOVESTATE_ABORT:
			fbMoveAxisABS.Execute := FALSE;
			fbMoveAxisABS2.Execute := FALSE;
			fbReset.Execute := FALSE;
			(* save target position*)
			rOldTargetPosition := 	q_stVGP.i_iPosition;
			fbHALT.Execute :=FALSE;
			fbPowerAxis.Enable := FALSE;
			fbPowerAxis.Enable_Positive := FALSE;
			fbPowerAxis.Enable_Negative := FALSE;
			q_stVGP.state := MOVESTATE_ENABLE; // Check homing first

	END_CASE





	
/// Motion Function Blocks
(* AXIS POWER*)
fbPowerAxis(
	Axis:= Axis, 
	Enable:= , 
	Enable_Positive:= , 
	Enable_Negative:= , 
	Override:= rOverride, 
	BufferMode:= , 
	Options:= , 
	Status=>  , 
	Busy=> PowerAxisOut.Busy , 
	Active=> PowerAxisOut.Active , 
	Error=> PowerAxisOut.Error, 
	ErrorID=> PowerAxisOut.ErrorID);
(* AXIS MOVE ABSOLUTE*)
fbMoveAxisABS(
	Axis:= Axis , 
	Execute:= , 
	Position:= , 
	Velocity:= , 
	Acceleration:= , 
	Deceleration:= , 
	Jerk:= , 
	BufferMode:= MC_BlendingNext , 
	Options:= , 
	Done=>MoveAbsoluteOut.Done, 
	Busy=> MoveAbsoluteOut.Busy, 
	Active=> MoveAbsoluteOut.Active, 
	CommandAborted=> MoveAbsoluteOut.CommandAborted , 
	Error=> MoveAbsoluteOut.Error, 
	ErrorID=> MoveAbsoluteOut.ErrorID);
	(* AXIS MOVE ABSOLUTE*)
fbMoveAxisABS2(
	Axis:= Axis , 
	Execute:= , 
	Position:= , 
	Velocity:= , 
	Acceleration:= , 
	Deceleration:= , 
	Jerk:= , 
	BufferMode:= MC_BlendingNext , 
	Options:= , 
	Done=>MoveAbsoluteOut2.Done, 
	Busy=> MoveAbsoluteOut2.Busy, 
	Active=> MoveAbsoluteOut2.Active, 
	CommandAborted=> MoveAbsoluteOut2.CommandAborted , 
	Error=> MoveAbsoluteOut2.Error, 
	ErrorID=> MoveAbsoluteOut2.ErrorID);
(*AXIS RESET*)
fbReset(
	Axis:= Axis, 
	Execute:= , 
	Done=>ResetOut.Done , 
	Busy=>ResetOut.Busy , 
	Error=> ResetOut.Error, 
	ErrorID=> ResetOut.ErrorID);
(*HALT*)
fbHalt(
	Axis:= Axis, 
	Execute:= , 
	Deceleration:= , 
	Jerk:= , 
	BufferMode:= MC_BlendingNext , 
	Options:= , 
	Done=> , 
	Busy=> , 
	Active=> , 
	CommandAborted=> , 
	Error=> , 
	ErrorID=> );
	

/// ERROR
IF Axis.Status.Error THEN
	q_stVGP.state := MOVESTATE_ERROR;	
END_IF;	
	
// Error Handling
if( fbPowerAxis.Error and fbPowerAxis.Active ) then 
	bError:= fbPowerAxis.Error;
	nErrorID:= fbPowerAxis.ErrorID;
END_IF
if( fbMoveAxisABS.Error and fbMoveAxisABS.Active ) then 
	bError:= fbMoveAxisABS.Error;
	nErrorID:= fbMoveAxisABS.ErrorID;
END_IF

(*Convert nErrorID to string*)
sErrorMessage:=WORD_TO_HEXSTR(in:=TO_WORD(nErrorID) , iPrecision:= 4, bLoCase:=0 );
END_ACTION

ACTION ACT_HOME:


CASE HomeState OF
	READY:
		fbSetPosition.Execute := FALSE;
		fbWriteParameter.Execute := FALSE;
		fbMoveRel.Execute := FALSE;
		
	INIT:
		// disable soft limits in order to be able to move the drive
		fbWriteParameter.ParameterNumber := MC_AxisParameter.EnableLimitNeg;//EnableLimitPos;// .EnableLimitNeg;
		fbWriteParameter.Value := FALSE;
		fbWriteParameter.Execute := TRUE;
		if (fbWriteParameter.Done) THEN
			fbWriteParameter.Execute := FALSE;
			HomeState:= MOVING; 
		END_IF

	MOVING:
		IF fbMoveRel.Done THEN
			fbMoveRel.Execute := TRUE;
		END_IF;
		IF fbMoveRel.Active  THEN
			(* axis is executing job but is not yet finished *)
			fbMoveRel.Execute := FALSE;
			HomeState := MOVING2;
		ElSIF fbMoveRel.Done THEN
			fbMoveRel.Execute := FALSE;
			HomeState := MOVING2;
		ELSIF fbMoveRel.CommandAborted OR fbMoveRel.Error THEN
			fbMoveRel.Execute := FALSE;
			HomeState := ERROR;
		END_IF
	
	MOVING2:
		IF fbMoveRel.Done THEN
			fbMoveRel.Execute := TRUE;
		END_IF;
		IF fbMoveRel.Active  THEN
			(* axis is executing job but is not yet finished *)
			fbMoveRel.Execute := FALSE;
			HomeState := MOVING;
		ElSIF fbMoveRel.Done THEN
			fbMoveRel.Execute := FALSE;
			HomeState := MOVING;
		ELSIF fbMoveRel.CommandAborted OR fbMoveRel.Error THEN
			fbMoveRel.Execute := FALSE;
			HomeState := CHECK;
		END_IF	

	
	CHECK:
		//Check position lag monitoring error
		if ( Axis.Status.ErrorID = 17245)THEN 
			// Set Current Position
			fbSetPosition.Position := 0; //rOpenPosition+rHomingDistance;
			fbSetPosition.Execute := TRUE;
			if ( fbSetPosition.Done ) THEN
				fbSetPosition.Execute := FALSE;
				HomeState:= WRITE;
			END_IF
		ELSE
			HomeState := ERROR;
		END_IF
	
	ERROR:
	
	
	WRITE:
	// Re Enable the Soft limits	
		fbWriteParameter.ParameterNumber := MC_AxisParameter.AxisEnMinSoftPosLimit;//AxisEnMaxSoftPosLimit;// .AxisEnMinSoftPosLimit;
		fbWriteParameter.Value := TRUE;
		fbWriteParameter.Execute := TRUE;
		if (fbWriteParameter.Done) THEN
			fbWriteParameter.Execute := FALSE;
			HomeState:= DONE; 
		END_IF
	
	DONE:
	// Homing DONE STATE 
	// should go back to closed zero position???

END_CASE

// Move Forward
fbMoveRel(
	Axis:= Axis , 
	Execute:= , 
	Distance:= rHomingDistance , 
	Velocity:= rHomingVelocity, 
	Acceleration:= , 
	Deceleration:= , 
	Jerk:= , 
	BufferMode:= MC_BlendingNext, 
	Options:= , 
	Done=> , 
	Busy=> , 
	Active=> , 
	CommandAborted=> , 
	Error=> , 
	ErrorID=> );
	
// Set Encoder Position
fbSetPosition(
	Axis:= Axis , 
	Execute:= , 
	Position:= 0 , 
	Mode:= , 
	Options:= , 
	Done=> , 
	Busy=> , 
	Error=> , 
	ErrorID=> );
	
// Write Parameters
fbWriteParameter(
	Axis:= Axis , 
	Execute:= , 
	ParameterNumber:= , 
	Value:= , 
	Done=> , 
	Busy=> , 
	Error=> , 
	ErrorID=> );
END_ACTION

ACTION ACT_INIT:
IF bInit THEN
	
(*
	(* init array with the interpolation points  *)
	(* 	fIn					 |		fOut		*)
	arrTable[1,1] := 0;			arrTable[1,2] := 0;
	arrTable[2,1] := 5;		    arrTable[2,2] := 135;
	arrTable[3,1] := 10;		arrTable[3,2] := 245;
	arrTable[4,1] :=  20;	    arrTable[4,2] := 405;
	arrTable[5,1] :=  30;	    arrTable[5,2] := 535;
	arrTable[6,1] := 40;		arrTable[6,2] := 689;
	arrTable[7,1] := 50;		arrTable[7,2] := 830;
	arrTable[8,1] := 60;	    arrTable[8,2] := 960;
	arrTable[9,1] := 70;	    arrTable[9,2] := 1095;
	arrTable[10,1] := 80;		arrTable[10,2] := 1225;
	arrTable[11,1] := 90;		arrTable[11,2] := 1415;
	arrTable[12,1] := 95;		arrTable[12,2] := 1495;
	arrTable[13,1] := 98;		arrTable[13,2] := 1559;
	arrTable[14,1] := 100;		arrTable[14,2] := 1645;
	*)
	
	(* init parameter struct *)
	stCTRL_LIN_INTERPOLATION_PARAMS.tCtrlCycleTime					:= T#10ms;
	stCTRL_LIN_INTERPOLATION_PARAMS.tTaskCycleTime					:= T#10ms;
	stCTRL_LIN_INTERPOLATION_PARAMS.nDataTable_NumberOfRows		:= INT_TO_UINT(14);

	(* set the addresses *)
	stCTRL_LIN_INTERPOLATION_PARAMS.pDataTable_ADR			:= ADR(arrTable);
	stCTRL_LIN_INTERPOLATION_PARAMS.nDataTable_SIZEOF		:= SIZEOF(arrTable);

	(* set the mode to ACTIVE --> normal operation *)
	eMode							:= eCTRL_MODE_ACTIVE;
	
	
	(* init array with the interpolation points  *)
	(* 	fIn					 |		fOut		*)
	 FOR iCounter:=1 TO 14 BY 1 DO
		arrTable_ENC[iCounter,1] := arrTable[iCounter,2];
		arrTable_ENC[iCounter,2] := arrTable[iCounter,1];		
	 END_FOR;
	(*
	arrTable_ENC[1,1] := 0;			arrTable_ENC[1,2] := 0;
	arrTable_ENC[2,1] := 135;		    arrTable_ENC[2,2] := 5;
	arrTable_ENC[3,1] := 245;		arrTable_ENC[3,2] := 10;
	arrTable_ENC[4,1] :=  405;	    arrTable_ENC[4,2] := 20;
	arrTable_ENC[5,1] :=  535;	    arrTable_ENC[5,2] := 30;
	arrTable_ENC[6,1] := 689;		arrTable_ENC[6,2] := 40;
	arrTable_ENC[7,1] := 830;		arrTable_ENC[7,2] := 50;
	arrTable_ENC[8,1] := 960;	    arrTable_ENC[8,2] := 60;
	arrTable_ENC[9,1] := 1095;	    arrTable_ENC[9,2] := 70;
	arrTable_ENC[10,1] := 1225;		arrTable_ENC[10,2] := 80;
	arrTable_ENC[11,1] := 1415;		arrTable_ENC[11,2] := 90;
	arrTable_ENC[12,1] := 1495;		arrTable_ENC[12,2] := 95;
	arrTable_ENC[13,1] := 1559;		arrTable_ENC[13,2] := 98;
	arrTable_ENC[14,1] := 1645;		arrTable_ENC[14,2] := 100;*)
	
	
	(* init parameter struct *)
	stCTRL_LIN_INTERPOLATION_PARAMS_ENC.tCtrlCycleTime					:= T#10ms;
	stCTRL_LIN_INTERPOLATION_PARAMS_ENC.tTaskCycleTime					:= T#10ms;
	stCTRL_LIN_INTERPOLATION_PARAMS_ENC.nDataTable_NumberOfRows		:= INT_TO_UINT(14);

	(* set the addresses *)
	stCTRL_LIN_INTERPOLATION_PARAMS_ENC.pDataTable_ADR			:= ADR(arrTable_ENC);
	stCTRL_LIN_INTERPOLATION_PARAMS_ENC.nDataTable_SIZEOF		:= SIZEOF(arrTable_ENC);
	
	(* reset the init flag *)
	bInit							:= FALSE;
	
END_IF;
END_ACTION

ACTION ACT_LIN_INTERPOLATION:

fbCTRL_LIN_INTERPOLATION(
	fIn:= q_stVGP.rReqPosition , 
	fManValue:= 0, 
	bExtrapolate:= , 
	eMode:= eMode, 
	fOut=> , 
	bInIsGreaterThanMaxElement=> , 
	bInIsLessThanMinElement=> , 
	eState=> , 
	eErrorId=> , 
	bError=> , 
	stParams:= stCTRL_LIN_INTERPOLATION_PARAMS );
	
// Target position Calculation
rTargetPosition := LREAL_TO_REAL(fbCTRL_LIN_INTERPOLATION.fOut);
//rTargetPosition := LIMIT(rClosePosition, rTargetPosition, rOpenPosition);	
	
fbCTRL_LIN_INTERPOLATION_ENC(
	fIn:= Axis.NcToPlc.ActPos , 
	fManValue:= 0, 
	bExtrapolate:= , 
	eMode:= eMode, 
	fOut=>  , 
	bInIsGreaterThanMaxElement=> , 
	bInIsLessThanMinElement=> , 
	eState=> , 
	eErrorId=> , 
	bError=> , 
	stParams:= stCTRL_LIN_INTERPOLATION_PARAMS_ENC );
q_stVGP.i_iPosition := LREAL_TO_REAL(fbCTRL_LIN_INTERPOLATION_ENC.fOut);
END_ACTION

METHOD ConfigEncoder : BOOL
VAR_INPUT
	EncoderMax: REAl; // Maximum encoder reading from fully closed to fully open
	invert: Bool; // Invert Encoder Counting Direction
END_VAR
VAR
	fbWriteParameter1: MC_WriteBoolParameter;
END_VAR
rOpenPosition := EncoderMax;

// fEncScaleFactor  -  AxisEncoderScalingFactor
 
// bEncIsInverse  -              
if (invert) THEN
	fbWriteParameter1.ParameterNumber :=  MC_AxisParameter.AxisEncoderDirectionInverse;
	fbWriteParameter1.Value := True;
END_IF

// Write Parameters
fbWriteParameter1(
	Axis:= Axis , 
	Execute:= , 
	ParameterNumber:= , 
	Value:= , 
	Done=> , 
	Busy=> , 
	Error=> , 
	ErrorID=> );
END_METHOD

METHOD M_INIT : BOOL
VAR_INPUT
	arrTable	: ARRAY[1..14,1..2] OF FLOAT;
	arrTable_ENC : ARRAY[1..14,1..2] OF FLOAT;
END_VAR
(* init array with the interpolation points  *)
	(* 	fIn					 |		fOut		*)
	arrTable[1,1] := 0;			arrTable[1,2] := 0;
	arrTable[2,1] := 5;		    arrTable[2,2] := 135;
	arrTable[3,1] := 10;		arrTable[3,2] := 245;
	arrTable[4,1] :=  20;	    arrTable[4,2] := 405;
	arrTable[5,1] :=  30;	    arrTable[5,2] := 535;
	arrTable[6,1] := 40;		arrTable[6,2] := 689;
	arrTable[7,1] := 50;		arrTable[7,2] := 830;
	arrTable[8,1] := 60;	    arrTable[8,2] := 960;
	arrTable[9,1] := 70;	    arrTable[9,2] := 1095;
	arrTable[10,1] := 80;		arrTable[10,2] := 1225;
	arrTable[11,1] := 90;		arrTable[11,2] := 1415;
	arrTable[12,1] := 95;		arrTable[12,2] := 1495;
	arrTable[13,1] := 98;		arrTable[13,2] := 1559;
	arrTable[14,1] := 100;		arrTable[14,2] := 1645;
	
	
	(* init parameter struct *)
	stCTRL_LIN_INTERPOLATION_PARAMS.tCtrlCycleTime					:= T#10ms;
	stCTRL_LIN_INTERPOLATION_PARAMS.tTaskCycleTime					:= T#10ms;
	stCTRL_LIN_INTERPOLATION_PARAMS.nDataTable_NumberOfRows		:= INT_TO_UINT(14);

	(* set the addresses *)
	stCTRL_LIN_INTERPOLATION_PARAMS.pDataTable_ADR			:= ADR(arrTable);
	stCTRL_LIN_INTERPOLATION_PARAMS.nDataTable_SIZEOF		:= SIZEOF(arrTable);

	(* set the mode to ACTIVE --> normal operation *)
	eMode							:= eCTRL_MODE_ACTIVE;
	
	
	(* init array with the interpolation points  *)
	(* 	fIn					 |		fOut		*)
	arrTable_ENC[1,1] := 0;			arrTable_ENC[1,2] := 0;
	arrTable_ENC[2,1] := 135;		    arrTable_ENC[2,2] := 5;
	arrTable_ENC[3,1] := 245;		arrTable_ENC[3,2] := 10;
	arrTable_ENC[4,1] :=  405;	    arrTable_ENC[4,2] := 20;
	arrTable_ENC[5,1] :=  535;	    arrTable_ENC[5,2] := 30;
	arrTable_ENC[6,1] := 689;		arrTable_ENC[6,2] := 40;
	arrTable_ENC[7,1] := 830;		arrTable_ENC[7,2] := 50;
	arrTable_ENC[8,1] := 960;	    arrTable_ENC[8,2] := 60;
	arrTable_ENC[9,1] := 1095;	    arrTable_ENC[9,2] := 70;
	arrTable_ENC[10,1] := 1225;		arrTable_ENC[10,2] := 80;
	arrTable_ENC[11,1] := 1415;		arrTable_ENC[11,2] := 90;
	arrTable_ENC[12,1] := 1495;		arrTable_ENC[12,2] := 95;
	arrTable_ENC[13,1] := 1559;		arrTable_ENC[13,2] := 98;
	arrTable_ENC[14,1] := 1645;		arrTable_ENC[14,2] := 100;
	
	
	(* init parameter struct *)
	stCTRL_LIN_INTERPOLATION_PARAMS_ENC.tCtrlCycleTime					:= T#10ms;
	stCTRL_LIN_INTERPOLATION_PARAMS_ENC.tTaskCycleTime					:= T#10ms;
	stCTRL_LIN_INTERPOLATION_PARAMS_ENC.nDataTable_NumberOfRows		:= INT_TO_UINT(14);

	(* set the addresses *)
	stCTRL_LIN_INTERPOLATION_PARAMS_ENC.pDataTable_ADR			:= ADR(arrTable_ENC);
	stCTRL_LIN_INTERPOLATION_PARAMS_ENC.nDataTable_SIZEOF		:= SIZEOF(arrTable_ENC);
END_METHOD

METHOD M_ValveControl : BOOL
VAR_INPUT
	state:E_VCN; // Close, Open, Pressure, Manual
END_VAR
q_stVGP.eValveControl := state;
END_METHOD

METHOD PUBLIC SetEncoderMax : BOOL
VAR_INPUT
	EncoderMax: REAl;
END_VAR
rOpenPosition := EncoderMax;
END_METHOD

END_FUNCTION_BLOCK

// ---- POUs/PRG_Gas_Selection.TcPOU
PROGRAM PRG_Gas_Selection
VAR
	CurrentGas: E_GasType;
	//pragma
	{attribute 'pytmc' := '
	pv: EM2K0:XGMD:GAS_TYPE ;
	type: mbbi ;
	field: ZRST none ;
	field: ONST Neon;
	field: TWST Argon ;
	field: THST Krypton ;
	field: FRST Xenon ;
	io: i
	'}
	SelectedGas: E_GasType;
END_VAR

(* Gas selection includes a purge and checks interlocks*)
//fix
if ( VVC_83.iq_stValve.q_xOPN_DO) then
	CurrentGas := E_GasType.Neon;
	elsif ( VVC_84.iq_stValve.q_xOPN_DO) then
		CurrentGas := E_GasType.Argon;
		elsif ( VVC_85.iq_stValve.q_xOPN_DO) then
		CurrentGas := E_GasType.Krypton;
			elsif ( VVC_86.iq_stValve.q_xOPN_DO) then
			CurrentGas := E_GasType.Xenon;
				else CurrentGas := E_GasType.none;
END_IF


If( CurrentGas <> SelectedGas) then
	bStartPurge_sw := true;
END_IF

if NOT(bStartPurge_sw) AND NOT(bPurgeActive)AND(bPurgeDone) then
	case SelectedGas of
	E_GasType.none: // all valves closed
		VVC_83.iq_stValve.pv_xOPN_SW:= false;
		VVC_84.iq_stValve.pv_xOPN_SW := false;
		VVC_85.iq_stValve.pv_xOPN_SW := false;
		VVC_86.iq_stValve.pv_xOPN_SW := false;
	E_GasType.Neon:
		VVC_83.iq_stValve.pv_xOPN_SW:= TRUE;
		VVC_84.iq_stValve.pv_xOPN_SW := false;
		VVC_85.iq_stValve.pv_xOPN_SW := false;
		VVC_86.iq_stValve.pv_xOPN_SW := false;
	E_GasType.Argon: // all valves closed
		VVC_83.iq_stValve.pv_xOPN_SW:= false;
		VVC_84.iq_stValve.pv_xOPN_SW := TRUE;
		VVC_85.iq_stValve.pv_xOPN_SW := false;
		VVC_86.iq_stValve.pv_xOPN_SW := false;	 
	E_GasType.Krypton: // all valves closed
		VVC_83.iq_stValve.pv_xOPN_SW:= false;
		VVC_84.iq_stValve.pv_xOPN_SW := false;
		VVC_85.iq_stValve.pv_xOPN_SW := TRUE;
		VVC_86.iq_stValve.pv_xOPN_SW := false;
	E_GasType.Xenon: // all valves closed
		VVC_83.iq_stValve.pv_xOPN_SW:= false;
		VVC_84.iq_stValve.pv_xOPN_SW := false;
		VVC_85.iq_stValve.pv_xOPN_SW := false;
		VVC_86.iq_stValve.pv_xOPN_SW := TRUE;
	END_CASE
END_IF


/// vcn and vgp on manual or auto??

END_PROGRAM

// ---- POUs/PRG_INJ.TcPOU
PROGRAM PRG_INJ
VAR
	i:INT;
	fullScale: REAL :=2000;
	DefaultSP :REAL:=0;
	rFULL_SCALE:REAL:=3000;//psig
END_VAR

// GCM
GCM_80(i_rFULL_SCALE := fullScale );
i:=i+1;
//GHC
GHC_50(PG=> );

// Vent Valves
// interlock evaluation

VVC_80.i_xExtILK_OK := true;//(NOT VVC_81.iq_stValve.q_xOPN_DO) AND(NOT VVC_82.iq_stValve.q_xOPN_DO); // Or we need to purge all the way up to the VCN
VVC_81.i_xExtILK_OK :=  (VVC_82.iq_stValve.q_xOPN_DO) AND(NOT VVC_83.iq_stValve.q_xOPN_DO) AND(NOT VVC_84.iq_stValve.q_xOPN_DO) AND (NOT VVC_85.iq_stValve.q_xOPN_DO) AND (NOT VVC_86.iq_stValve.q_xOPN_DO);// AND (NOT VVC_80.iq_stValve.q_xOPN_DO);
VVC_82.i_xExtILK_OK := (NOT VVC_83.iq_stValve.q_xOPN_DO) AND(NOT VVC_84.iq_stValve.q_xOPN_DO) AND (NOT VVC_85.iq_stValve.q_xOPN_DO) AND (NOT VVC_86.iq_stValve.q_xOPN_DO);// AND (NOT VVC_80.iq_stValve.q_xOPN_DO);

// instanitation
VVC_80(i_xExtILK_OK:= , i_xOverrideMode:= xOverrideMode, iq_stValve=> );
VVC_81(i_xExtILK_OK:= , i_xOverrideMode:= xOverrideMode, iq_stValve=> );
VVC_82(i_xExtILK_OK:= , i_xOverrideMode:= xOverrideMode, iq_stValve=> );



// Gas panel

// Interlock evaluation
VVC_83.i_xExtILK_OK := (NOT VVC_84.iq_stValve.q_xOPN_DO) AND (NOT VVC_85.iq_stValve.q_xOPN_DO) AND (NOT VVC_86.iq_stValve.q_xOPN_DO) AND (NOT VVC_81.iq_stValve.q_xOPN_DO) AND (NOT VVC_82.iq_stValve.q_xOPN_DO) AND NOT bPurgeActive;  
VVC_84.i_xExtILK_OK := (NOT VVC_83.iq_stValve.q_xOPN_DO) AND (NOT VVC_85.iq_stValve.q_xOPN_DO) AND (NOT VVC_86.iq_stValve.q_xOPN_DO) AND (NOT VVC_81.iq_stValve.q_xOPN_DO) AND (NOT VVC_82.iq_stValve.q_xOPN_DO) AND NOT bPurgeActive  ;
VVC_85.i_xExtILK_OK := (NOT VVC_83.iq_stValve.q_xOPN_DO) AND (NOT VVC_84.iq_stValve.q_xOPN_DO) AND (NOT VVC_86.iq_stValve.q_xOPN_DO) AND (NOT VVC_81.iq_stValve.q_xOPN_DO) AND (NOT VVC_82.iq_stValve.q_xOPN_DO) AND NOT bPurgeActive;  
VVC_86.i_xExtILK_OK := (NOT VVC_83.iq_stValve.q_xOPN_DO) AND (NOT VVC_84.iq_stValve.q_xOPN_DO) AND (NOT VVC_85.iq_stValve.q_xOPN_DO) AND (NOT VVC_81.iq_stValve.q_xOPN_DO) AND (NOT VVC_82.iq_stValve.q_xOPN_DO) AND NOT bPurgeActive ;

//Gas Panel
VVC_83(i_xExtILK_OK:= , i_xOverrideMode:= xOverrideMode, iq_stValve=> );
VVC_84(i_xExtILK_OK:= , i_xOverrideMode:= xOverrideMode, iq_stValve=> );
VVC_85(i_xExtILK_OK:= , i_xOverrideMode:= xOverrideMode, iq_stValve=> );
VVC_86(i_xExtILK_OK:= , i_xOverrideMode:= xOverrideMode, iq_stValve=> );

END_PROGRAM

// ---- POUs/PRG_Purge.TcPOU
PROGRAM PRG_Purge
VAR
	step: INT:=0;

//ADD PRAGMAS

	AllGasVlvCls 		: BOOL; (* All Gas Manifold Valves are closed when True, not including VIC80, 81 or VGP40 *)
	WatchdogTmr			: TON;  (* Purge Watchdog Timer*)

	StartWatchdogTmr 	: BOOL;
	WatchdogPeriod 		: TIME;

	NeedleVlvPurgeTmr	: TON;	(* Declaration for the needle valve Purge timer *)
	tNeedlePurgeTime		: TIME:=T#30S;
	BurpET				: TIME;
	NeedlePurgeRun		: BOOL;
	NeedlePurgeDone		: BOOL;
	NeedlePurgeRepeat	: INT:= 2;
	VCN_Timer	:TON;
	


	//PRAGMA
	GBA80Tmr			: TON;
	GBA80Time			: TIME:=T#20S;
	GBATimeDone			: BOOL;

	CATCH : INT;
	CATCH1 : INT;
	
	// Timers
	VVC_81_Timer : TON;
	VVC_82_Timer : TON;
	VVC_81_Time			: TIME:=T#60S;
	VVC_82_Time			: TIME:=T#120S;
	
	
	

END_VAR


(* 		PURGE CYCLE
	The purge cycle cosists of the following steps;	
	1. Close all gas valves 83-86
	2. Close Needle valve 
	3. Fully open VGP:40
	4. PUMP DOWN MANIFOLD: Open VIC82 for a certain peroid of time or till cetrain pressure
	5. Open VIC:81 and keep it open while the manifold pumps down to pressure set point
	6. BURP NEEDLE VALVE: Once the manifold is pumped down, open the needle valve (burp) to evacuate gases that may be trapped in its mechanism
	7. Close needle valve
	8. Close VIC:81 and VIC:82
	9. Release VGP:40

*)
tNeedlePurgeTime := INT_TO_TIME(iNeedleBurpTIME);

CASE step OF
		0: // READY STATE
		IF (bStartPurge_sw) Then
			step:=10;
			bPurgeActive := TRUE;
			bPurgeDone := FALSE;
		END_IF

10: // start purge sequence by closing all gas valves
	VVC_80.M_Set_OPN_SW(false);
	VVC_83.M_Set_OPN_SW(false);
	VVC_84.M_Set_OPN_SW(false);
	VVC_85.M_Set_OPN_SW(false);
	VVC_86.M_Set_OPN_SW(false);
	
	if  (NOT VVC_83.iq_stValve.q_xOPN_DO) AND (NOT VVC_83.iq_stValve.q_xOPN_DO) AND(NOT VVC_84.iq_stValve.q_xOPN_DO) AND (NOT VVC_85.iq_stValve.q_xOPN_DO) AND (NOT VVC_86.iq_stValve.q_xOPN_DO) then
		step:= 20;
	END_IF
	
20: //Close Needle valve 
	VCN_50.M_ValveControl(E_VCN.CloseValve);
	// wait for a period of time to ensure that the Valve is fully closed
	IF (VCN_Timer.Q) THEN
		step:=30;
	END_IF
	
	
30: //Fully open VGP:40
	VGP_50.M_ValveControl(E_VCN.OpenValve); 
	IF NOT(VGP_50.q_stVGP.state = E_MoveState.MOVESTATE_READY ) THEN // wait until the VGP encoder reads Open
		step:=31;
	END_IF
	if (VGP_50.q_stVGP.pv_xError )then
		step:=900+step;
	END_IF
31: 
	IF (VGP_50.q_stVGP.state = E_MoveState.MOVESTATE_READY ) THEN // wait until the VGP encoder reads Open //use motion ready
		step:=40;
	END_IF
	if (VGP_50.q_stVGP.pv_xError )then
		step:=900+step;
	END_IF
	
40: // open vavle 80 to pump down all the way to the needle valve
	VVC_80.M_Set_OPN_SW(TRUE);
	if (VVC_80.iq_stValve.q_xOPN_DO ) THEN
		step:=41;
	END_IF


41 :  //PUMP DOWN MANIFOLD: Open VIC82 for a certain peroid of time or till cetrain pressure
	VVC_82.M_Set_OPN_SW(TRUE);
	if (VVC_82.iq_stValve.q_xOPN_DO ) AND (VVC_82_Timer.Q) THEN
		step:=50;
	END_IF

50:// Open VIC:81 and keep it open while the manifold pumps down to pressure set point
	VVC_81.M_Set_OPN_SW(TRUE);
	IF (VVC_81.iq_stValve.q_xOPN_DO ) AND (VVC_81_Timer.Q) THEN // or a certain pressure reading and check timeouts
		step:=51;
	END_IF

51://Close VIC:80 VIC:81 and VIC:82
	VVC_80.M_Set_OPN_SW(false);
	VVC_81.M_Set_OPN_SW(false);
	VVC_82.M_Set_OPN_SW(false);
	
	IF (NOT VVC_80.iq_stValve.q_xOPN_DO) AND (NOT VVC_81.iq_stValve.q_xOPN_DO) AND(NOT VVC_82.iq_stValve.q_xOPN_DO) THEN
		step:=60;
	END_IF

60: //BURP NEEDLE VALVE: Once the manifold is pumped down, open the needle valve (burp) to evacuate gases that may be trapped in its mechanism
	VCN_50.M_ValveControl(E_VCN.OpenValve); 
	// wait for a period of time to ensure that the Valve is fully open
	IF (VCN_Timer.Q) THEN
		step:=70;
	END_IF

70: //Close Needle valve 
	VCN_50.M_ValveControl(E_VCN.CloseValve);
	// wait for a period of time to ensure that the Valve is fully closed
	IF (VCN_Timer.Q) THEN
		step:=80;
	END_IF

80: // Repeat
	IF (NeedlePurgeRepeat > 0) THEN
		NeedlePurgeRepeat := NeedlePurgeRepeat-1;
		step:= 60;
	ELSE
		NeedlePurgeRepeat := 2;
		step:=90;				
	END_IF
	
	

90: //Release VGP:40
	VGP_50.M_ValveControl(E_VCN.ManualControl);
	VGP_50.q_stVGP.rReqPosition:= 50; //50% open
	IF NOT(VGP_50.q_stVGP.state = E_MoveState.MOVESTATE_READY ) THEN // wait until the VGP encoder reads Open //use motion ready
		step:=91;
	END_IF
	if (VGP_50.q_stVGP.pv_xError )then
		step:=900+step;
	END_IF
	
91: 
	IF (VGP_50.q_stVGP.state = E_MoveState.MOVESTATE_READY ) THEN // wait until the VGP encoder reads Open //use motion ready
		step:=100;
	END_IF
	if (VGP_50.q_stVGP.pv_xError )then
		step:=900+step;
	END_IF
  
100: // DONE
	bStartPurge_sw := false;
	bPurgeActive := false;
	bPurgeDone := TRUE;
	
900: //Error
	VVC_80.M_Set_OPN_SW(false);
	VVC_81.M_Set_OPN_SW(false);
	VVC_82.M_Set_OPN_SW(false);
	VVC_83.M_Set_OPN_SW(false);
	VVC_84.M_Set_OPN_SW(false);
	VVC_85.M_Set_OPN_SW(false);
	VVC_86.M_Set_OPN_SW(false);
	VCN_50.M_ValveControl(E_VCN.CloseValve);
	//VGP_50.M_ValveControl(E_VCN.CloseValve); // CLOSE or OPEN to pump down

END_CASE


//shouldn't be here
(*
if (bPurgeActive) then
	VVC_83.i_xExtILK_OK := VVC_84.i_xExtILK_OK := VVC_85.i_xExtILK_OK := VVC_86.i_xExtILK_OK := false;
END_IF
*)

//Errors
if (step >900 ) Then
	// show error and step
END_IF


//Timers
VVC_81_Timer(IN:= (step = 50), PT:=VVC_81_Time);
VVC_82_Timer(IN:= (step = 41), PT:=VVC_82_Time);
VCN_Timer(IN:= (step = 20) OR (step = 60) OR (step = 70), PT:=tNeedlePurgeTime);


/// vcn and vgp on manual or auto?? manual, until the Go or auto button is pressed??

END_PROGRAM

// ---- POUs/PRG_VGP.TcPOU
PROGRAM PRG_VGP
VAR
	arrTable											: ARRAY[1..14,1..2] OF FLOAT;
	arrTable_ENC										: ARRAY[1..14,1..2] OF FLOAT;
	
	bInit: BOOL:=true;
	
	VGP_REQ_POS: LREAL;
	VGP_OUT_POS:LREAL;
END_VAR


IF bInit
THEN
	
	
	(* init array with the interpolation points  *)
	(* 	fIn					 |		fOut		*)
	arrTable[1,1] := 0;			arrTable[1,2] := 0;
	arrTable[2,1] := 5;		    arrTable[2,2] := 170;
	arrTable[3,1] := 10;		arrTable[3,2] := 280;
	arrTable[4,1] :=  20;	    arrTable[4,2] := 445;
	arrTable[5,1] :=  30;	    arrTable[5,2] := 575;
	arrTable[6,1] := 40;		arrTable[6,2] := 725;
	arrTable[7,1] := 50;		arrTable[7,2] := 860;
	arrTable[8,1] := 60;	    arrTable[8,2] := 980;
	arrTable[9,1] := 70;	    arrTable[9,2] := 1120;
	arrTable[10,1] := 80;		arrTable[10,2] := 1250;
	arrTable[11,1] := 90;		arrTable[11,2] := 1420;
	arrTable[12,1] := 95;		arrTable[12,2] := 1550;
	arrTable[13,1] := 98;		arrTable[13,2] := 1600;
	arrTable[14,1] := 100;		arrTable[14,2] := 1660;
	
	
	(* reset the init flag *)
	bInit							:= FALSE;
END_IF

VGP_50.i_xOpenIlkOK := (fb_EM2K0_XGMD_PTM_50.iq_stPtm.eState = pumpRUNNING) ;
 
VGP_50(
	i_xExtIlkOK:=(fb_EM2K0_XGMD_PTM_50.iq_stPtm.eState = pumpRUNNING), 
	i_ReqPos:=  , 
	arrTable:= arrTable , 
	(*arrTable_ENC:= arrTable_ENC , *)
	q_stVGP=> );

END_PROGRAM
